(* Logix 5000 project; controller LeakTestAuto vendor 1 type 14 code 226 rev 37.11; software revision 37.01; part 7 of 13 *)
(* tags used below, declared in another part *)
   AOI_CTS1 : AOI_CTS_INSTRUMENT;
   AOI_CTS2 : AOI_CTS_INSTRUMENT;
   AOI_RobotPos : AOI_RobotPositions;
   AOI_SeqSteps : AOI_StandardSeqSteps;
   Conveyor : udt_OutputStructure;
   Conveyor_Seq : udt_SequenceStructure_X64;
   CurrentDUTData : udt_DUTHistory[2];
   DryCycle_N1Ready : BOOL;
   DryCycle_N2Ready : BOOL;
   DUTHistoryDump : udt_DUTHistory;
   DUTTestHistory : udt_DUTHistory[10];
   FFLU_DUTHistory : CONTROL;
   LeakTester1 : udt_OutputStructure;
   LeakTester2 : udt_OutputStructure;
   Nest2Cylinder : udt_OutputStructure;
   OP220 : udt_Mode;
   OP220_Seq : udt_SequenceStructure_X64;
   OutfeedCounter : COUNTER;
   Robot : udt_OutputStructure;
   RobotGripper : udt_OutputStructure;
   RobotInputs : udt_EpsonInputs;
   TON_FailChute : TIMER[10];
   Delay_TMR : TIMER[11];   // Delay Timers
   I_OP220_N3_CONVEYOR_LOAD : ALIAS FOR Local:3:I.Pt12.Data;
   I_OP220_N3_DUT_PRE_NEST_1 : ALIAS FOR Local:3:I.Pt01.Data;
   I_OP220_N3_DUT_PRE_NEST_2 : ALIAS FOR Local:3:I.Pt02.Data;
   I_OP220_N3_NEST2_EXTEND : ALIAS FOR Local:3:I.Pt06.Data;
   I_OP220_N3_REJECT_BIN_OK : ALIAS FOR Local:3:I.Pt09.Data;
   I_OP220_N3_REJECT_CHUTE_PART : ALIAS FOR Local:3:I.Pt10.Data;
   Ignition_Bypass : BOOL;
   James_Dint : DINT;   // James Test Word
   null : STRING;
   ST1_Ignition_DataReady : BOOL;
   ST1_Ignition_DataReady_Setup : BOOL;
   ST1_Ignition_DataReceived : BOOL;
   ST1_Ignition_SerialNum : STRING;
   ST1_Ignition_Status : DINT;
   ST2_Ignition_DataReady : BOOL;
   ST2_Ignition_DataReady_Setup : BOOL;
   ST2_Ignition_DataReceived : BOOL;
   ST2_Ignition_SerialNum : STRING;
   ST2_Ignition_Status : DINT;
(* MainProgram, continued *)

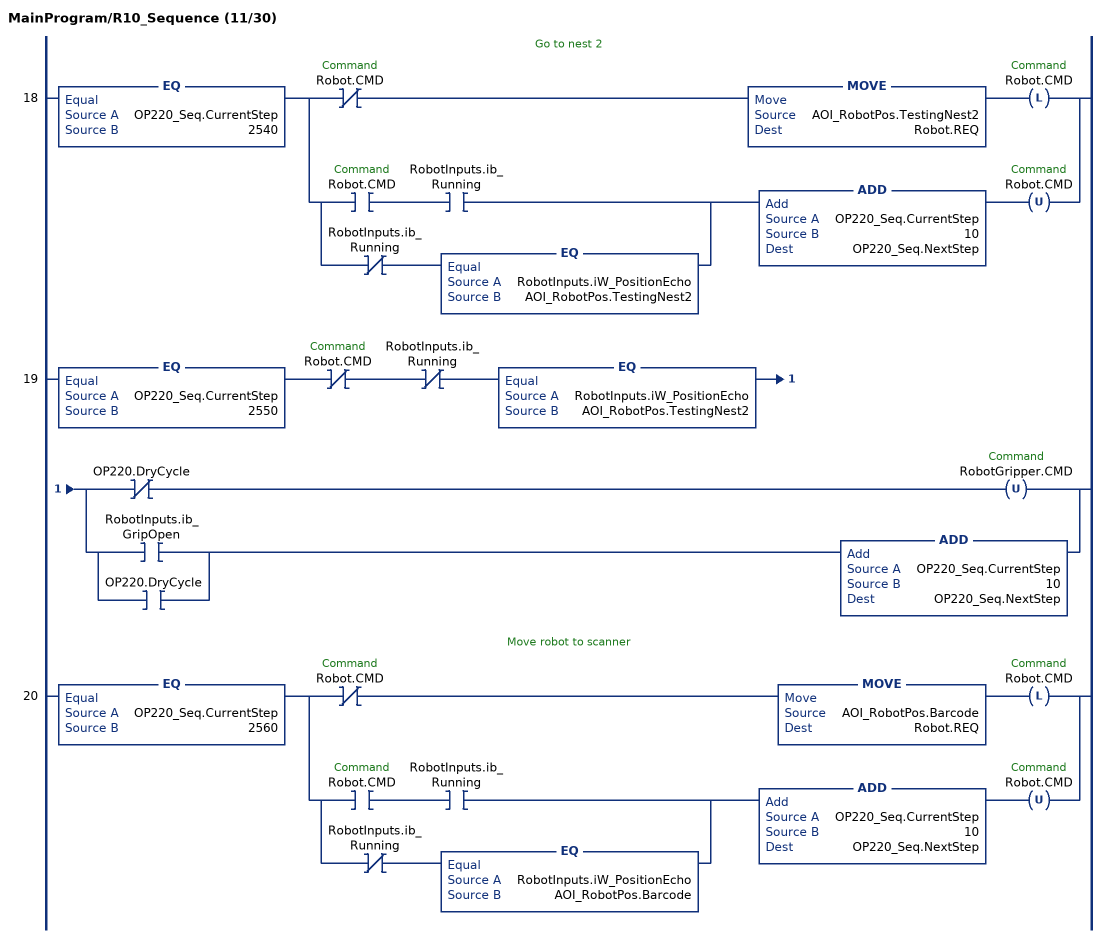
   [picture p74: MainProgram/R10_Sequence rungs 18-20]
   // Go to nest 2
   18: EQ(OP220_Seq.CurrentStep,2540)[XIO(Robot.CMD) MOVE(AOI_RobotPos.TestingNest2,Robot.REQ) OTL(Robot.CMD) ,[XIC(Robot.CMD) XIC(RobotInputs.ib_Running) ,XIO(RobotInputs.ib_Running) EQ(RobotInputs.iW_PositionEcho,AOI_RobotPos.TestingNest2) ] ADD(OP220_Seq.CurrentStep,10,OP220_Seq.NextStep) OTU(Robot.CMD) ];
   19: EQ(OP220_Seq.CurrentStep,2550)XIO(Robot.CMD)XIO(RobotInputs.ib_Running)EQ(RobotInputs.iW_PositionEcho,AOI_RobotPos.TestingNest2)[XIO(OP220.DryCycle) OTU(RobotGripper.CMD) ,[XIC(RobotInputs.ib_GripOpen) ,XIC(OP220.DryCycle) ] ADD(OP220_Seq.CurrentStep,10,OP220_Seq.NextStep) ];
   // Move robot to scanner
   20: EQ(OP220_Seq.CurrentStep,2560)[XIO(Robot.CMD) MOVE(AOI_RobotPos.Barcode,Robot.REQ) OTL(Robot.CMD) ,[XIC(Robot.CMD) XIC(RobotInputs.ib_Running) ,XIO(RobotInputs.ib_Running) EQ(RobotInputs.iW_PositionEcho,AOI_RobotPos.Barcode) ] ADD(OP220_Seq.CurrentStep,10,OP220_Seq.NextStep) OTU(Robot.CMD) ];
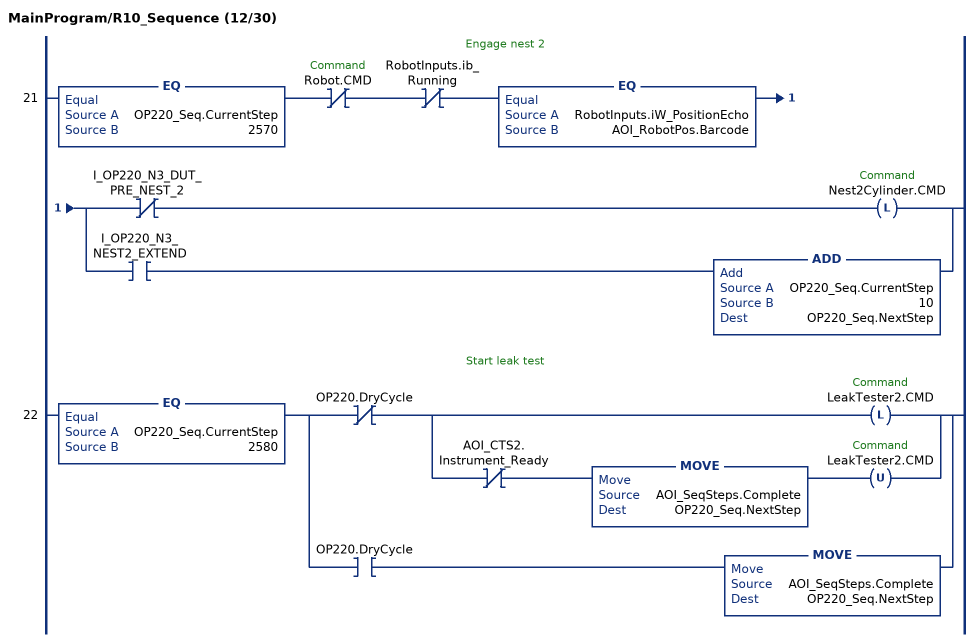
   // Engage nest 2
   21: EQ(OP220_Seq.CurrentStep,2570)XIO(Robot.CMD)XIO(RobotInputs.ib_Running)EQ(RobotInputs.iW_PositionEcho,AOI_RobotPos.Barcode)[XIO(I_OP220_N3_DUT_PRE_NEST_2) OTL(Nest2Cylinder.CMD) ,XIC(I_OP220_N3_NEST2_EXTEND) ADD(OP220_Seq.CurrentStep,10,OP220_Seq.NextStep) ];
   // Start leak test
   22: EQ(OP220_Seq.CurrentStep,2580)[XIO(OP220.DryCycle) [OTL(LeakTester2.CMD) ,XIO(AOI_CTS2.Instrument_Ready) MOVE(AOI_SeqSteps.Complete,OP220_Seq.NextStep) OTU(LeakTester2.CMD) ] ,XIC(OP220.DryCycle) MOVE(AOI_SeqSteps.Complete,OP220_Seq.NextStep) ];
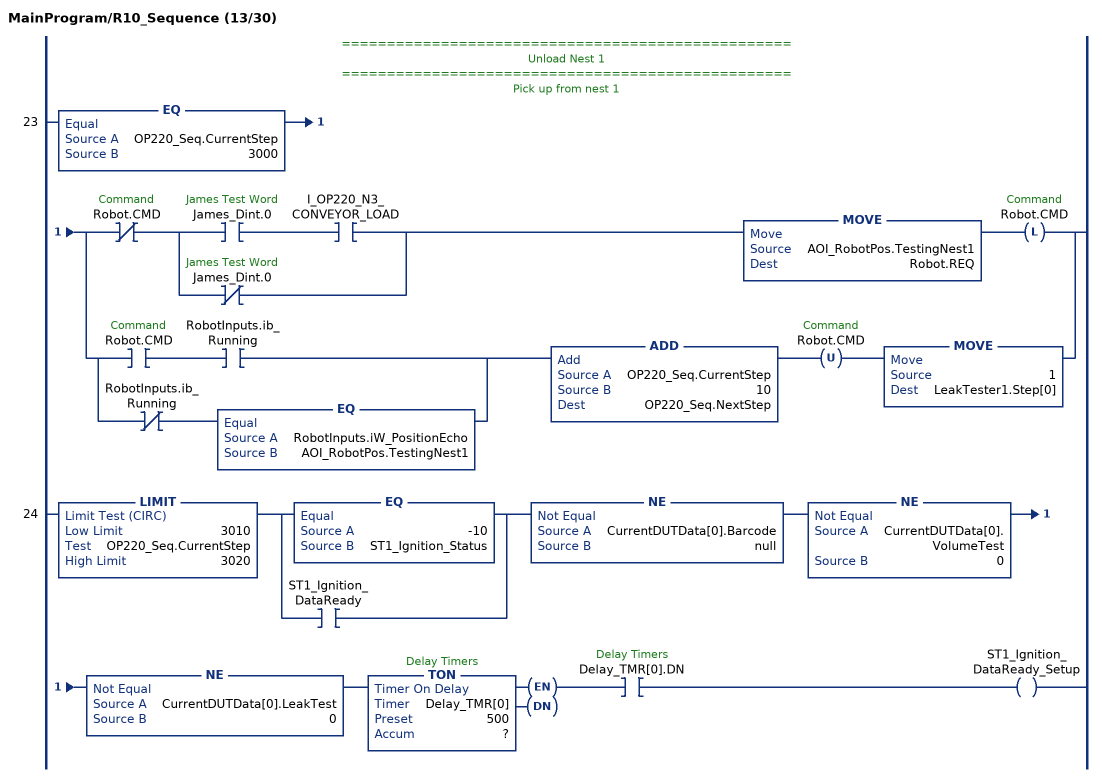
   // ==================================================
   // Unload Nest 1
   // ==================================================
   // Pick up from nest 1
   23: EQ(OP220_Seq.CurrentStep,3000)[XIO(Robot.CMD) [XIC(James_Dint.0) XIC(I_OP220_N3_CONVEYOR_LOAD) ,XIO(James_Dint.0) ] MOVE(AOI_RobotPos.TestingNest1,Robot.REQ) OTL(Robot.CMD) ,[XIC(Robot.CMD) XIC(RobotInputs.ib_Running) ,XIO(RobotInputs.ib_Running) EQ(RobotInputs.iW_PositionEcho,AOI_RobotPos.TestingNest1) ] ADD(OP220_Seq.CurrentStep,10,OP220_Seq.NextStep) OTU(Robot.CMD) MOVE(1,LeakTester1.Step[0]) ];
   24: LIMIT(3010,OP220_Seq.CurrentStep,3020)[EQ(-10,ST1_Ignition_Status) ,XIC(ST1_Ignition_DataReady) ]NE(CurrentDUTData[0].Barcode,null)NE(CurrentDUTData[0].VolumeTest,0)NE(CurrentDUTData[0].LeakTest,0)TON(Delay_TMR[0],?,?)XIC(Delay_TMR[0].DN)OTE(ST1_Ignition_DataReady_Setup);
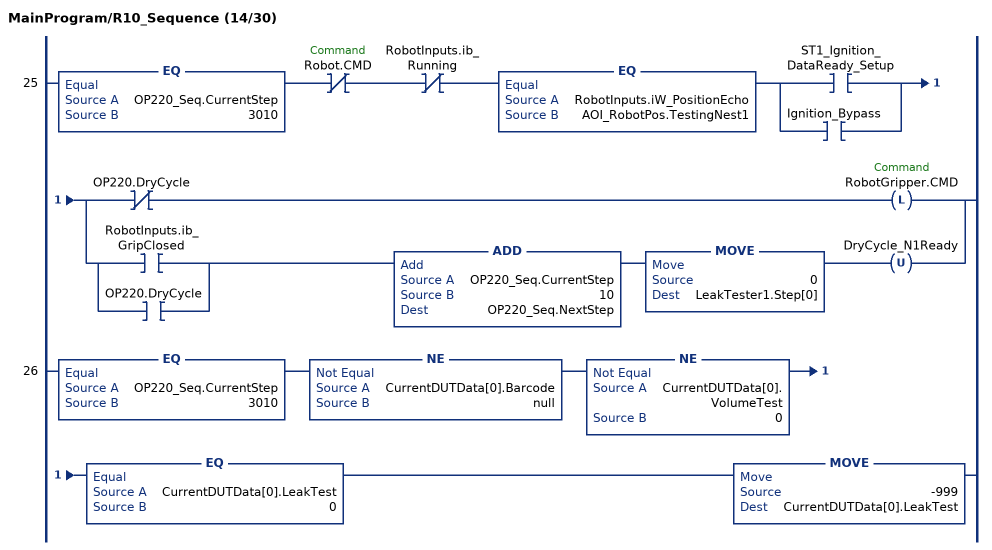
   25: EQ(OP220_Seq.CurrentStep,3010)XIO(Robot.CMD)XIO(RobotInputs.ib_Running)EQ(RobotInputs.iW_PositionEcho,AOI_RobotPos.TestingNest1)[XIC(ST1_Ignition_DataReady_Setup) ,XIC(Ignition_Bypass) ][XIO(OP220.DryCycle) OTL(RobotGripper.CMD) ,[XIC(RobotInputs.ib_GripClosed) ,XIC(OP220.DryCycle) ] ADD(OP220_Seq.CurrentStep,10,OP220_Seq.NextStep) MOVE(0,LeakTester1.Step[0]) OTU(DryCycle_N1Ready) ];
   26: EQ(OP220_Seq.CurrentStep,3010)NE(CurrentDUTData[0].Barcode,null)NE(CurrentDUTData[0].VolumeTest,0)EQ(CurrentDUTData[0].LeakTest,0)MOVE(-999,CurrentDUTData[0].LeakTest);
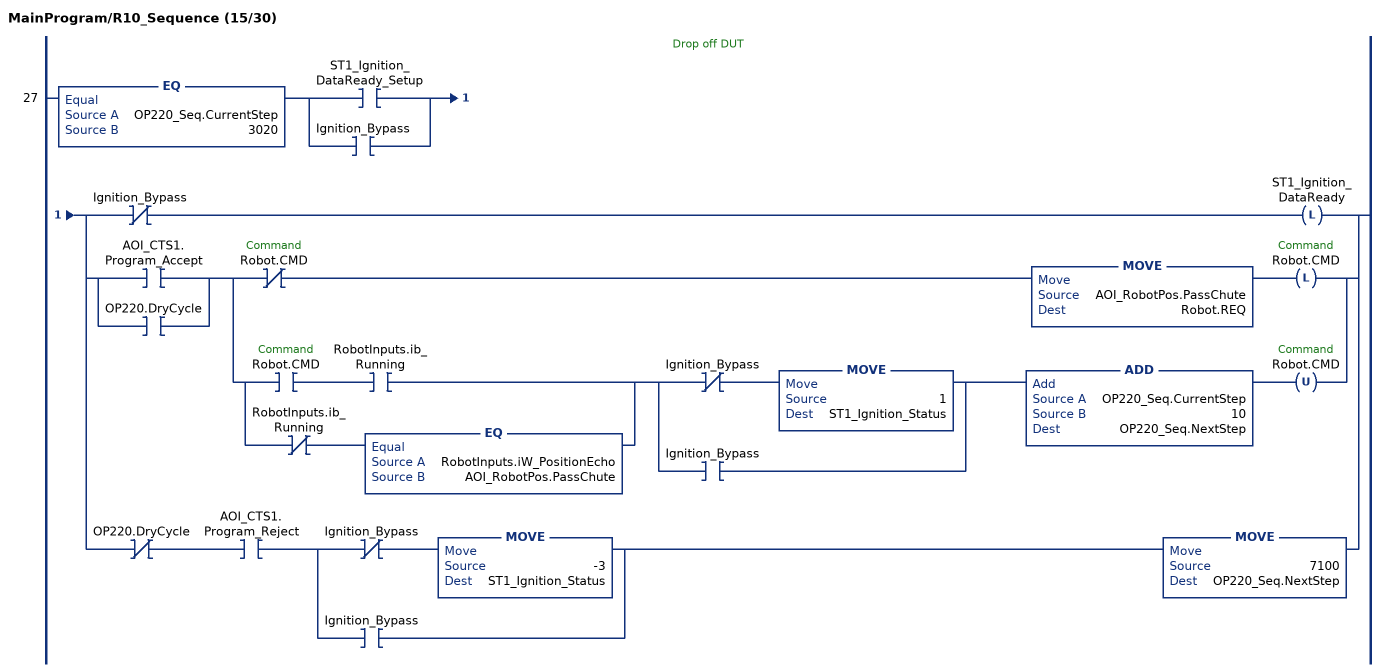
   // Drop off DUT
   27: EQ(OP220_Seq.CurrentStep,3020)[XIC(ST1_Ignition_DataReady_Setup) ,XIC(Ignition_Bypass) ][XIO(Ignition_Bypass) OTL(ST1_Ignition_DataReady) ,[XIC(AOI_CTS1.Program_Accept) ,XIC(OP220.DryCycle) ] [XIO(Robot.CMD) MOVE(AOI_RobotPos.PassChute,Robot.REQ) OTL(Robot.CMD) ,[XIC(Robot.CMD) XIC(RobotInputs.ib_Running) ,XIO(RobotInputs.ib_Running) EQ(RobotInputs.iW_PositionEcho,AOI_RobotPos.PassChute) ] [XIO(Ignition_Bypass) MOVE(1,ST1_Ignition_Status) ,XIC(Ignition_Bypass) ] ADD(OP220_Seq.CurrentStep,10,OP220_Seq.NextStep) OTU(Robot.CMD) ] ,XIO(OP220.DryCycle) XIC(AOI_CTS1.Program_Reject) [XIO(Ignition_Bypass) MOVE(-3,ST1_Ignition_Status) ,XIC(Ignition_Bypass) ] MOVE(7100,OP220_Seq.NextStep) ];
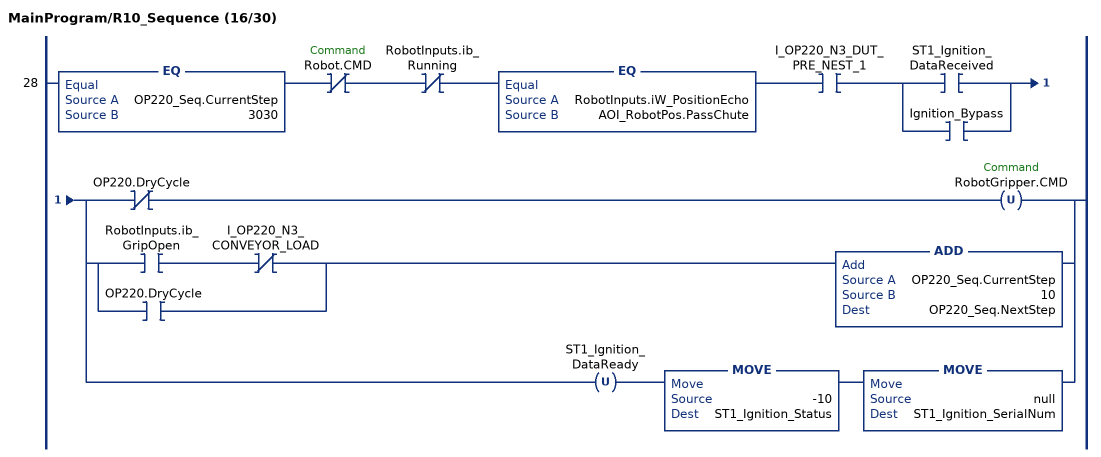
   28: EQ(OP220_Seq.CurrentStep,3030)XIO(Robot.CMD)XIO(RobotInputs.ib_Running)EQ(RobotInputs.iW_PositionEcho,AOI_RobotPos.PassChute)XIC(I_OP220_N3_DUT_PRE_NEST_1)[XIC(ST1_Ignition_DataReceived) ,XIC(Ignition_Bypass) ][XIO(OP220.DryCycle) OTU(RobotGripper.CMD) ,[XIC(RobotInputs.ib_GripOpen) XIO(I_OP220_N3_CONVEYOR_LOAD) ,XIC(OP220.DryCycle) ] ADD(OP220_Seq.CurrentStep,10,OP220_Seq.NextStep) ,OTU(ST1_Ignition_DataReady) MOVE(-10,ST1_Ignition_Status) MOVE(null,ST1_Ignition_SerialNum) ];
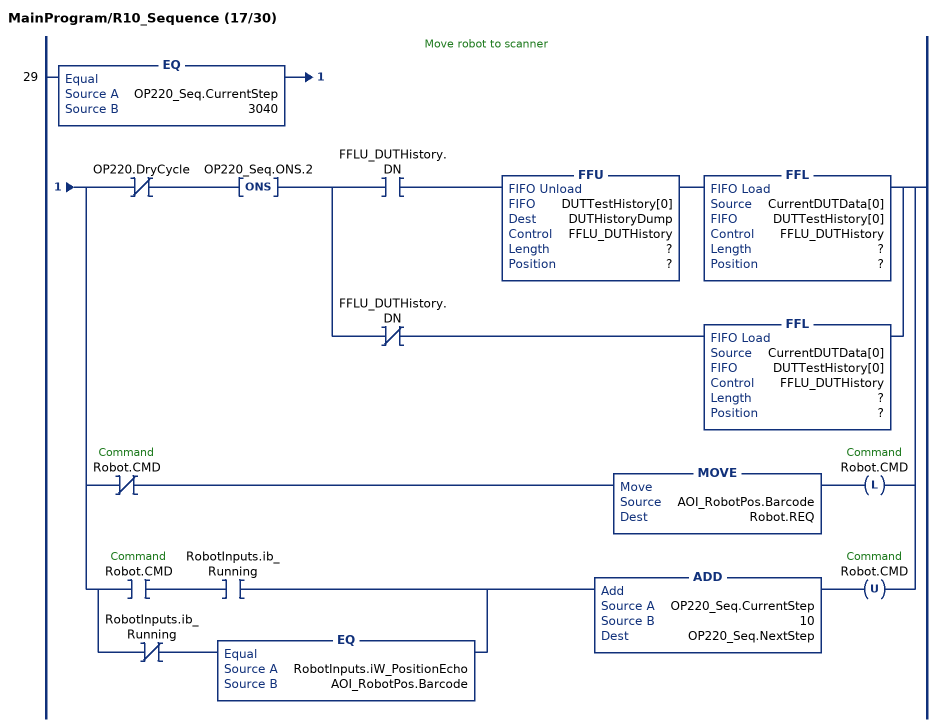
   // Move robot to scanner
   29: EQ(OP220_Seq.CurrentStep,3040)[XIO(OP220.DryCycle) ONS(OP220_Seq.ONS.2) [XIC(FFLU_DUTHistory.DN) FFU(DUTTestHistory[0],DUTHistoryDump,FFLU_DUTHistory,?,?) FFL(CurrentDUTData[0],DUTTestHistory[0],FFLU_DUTHistory,?,?) ,XIO(FFLU_DUTHistory.DN) FFL(CurrentDUTData[0],DUTTestHistory[0],FFLU_DUTHistory,?,?) ] ,XIO(Robot.CMD) MOVE(AOI_RobotPos.Barcode,Robot.REQ) OTL(Robot.CMD) ,[XIC(Robot.CMD) XIC(RobotInputs.ib_Running) ,XIO(RobotInputs.ib_Running) EQ(RobotInputs.iW_PositionEcho,AOI_RobotPos.Barcode) ] ADD(OP220_Seq.CurrentStep,10,OP220_Seq.NextStep) OTU(Robot.CMD) ];
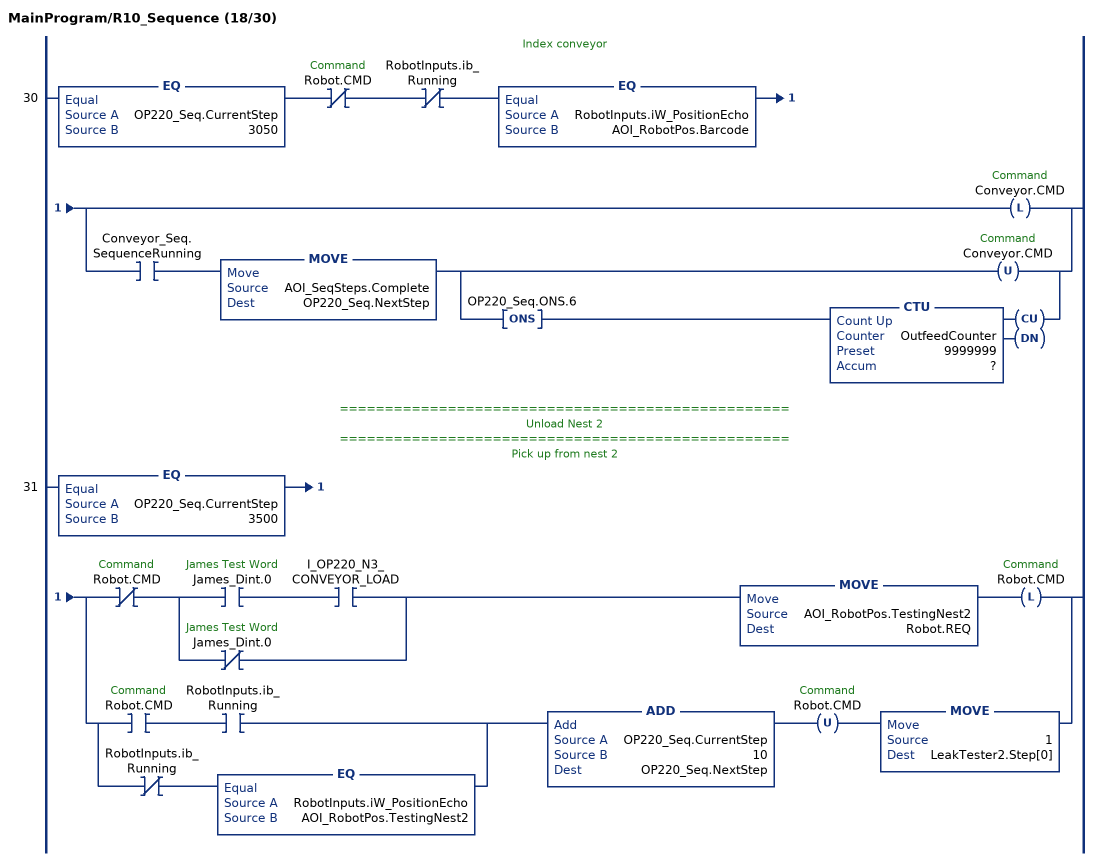
   // Index conveyor
   30: EQ(OP220_Seq.CurrentStep,3050)XIO(Robot.CMD)XIO(RobotInputs.ib_Running)EQ(RobotInputs.iW_PositionEcho,AOI_RobotPos.Barcode)[OTL(Conveyor.CMD) ,XIC(Conveyor_Seq.SequenceRunning) MOVE(AOI_SeqSteps.Complete,OP220_Seq.NextStep) [OTU(Conveyor.CMD) ,ONS(OP220_Seq.ONS.6) CTU(OutfeedCounter,?,?) ] ];
   // ==================================================
   // Unload Nest 2
   // ==================================================
   // Pick up from nest 2
   31: EQ(OP220_Seq.CurrentStep,3500)[XIO(Robot.CMD) [XIC(James_Dint.0) XIC(I_OP220_N3_CONVEYOR_LOAD) ,XIO(James_Dint.0) ] MOVE(AOI_RobotPos.TestingNest2,Robot.REQ) OTL(Robot.CMD) ,[XIC(Robot.CMD) XIC(RobotInputs.ib_Running) ,XIO(RobotInputs.ib_Running) EQ(RobotInputs.iW_PositionEcho,AOI_RobotPos.TestingNest2) ] ADD(OP220_Seq.CurrentStep,10,OP220_Seq.NextStep) OTU(Robot.CMD) MOVE(1,LeakTester2.Step[0]) ];
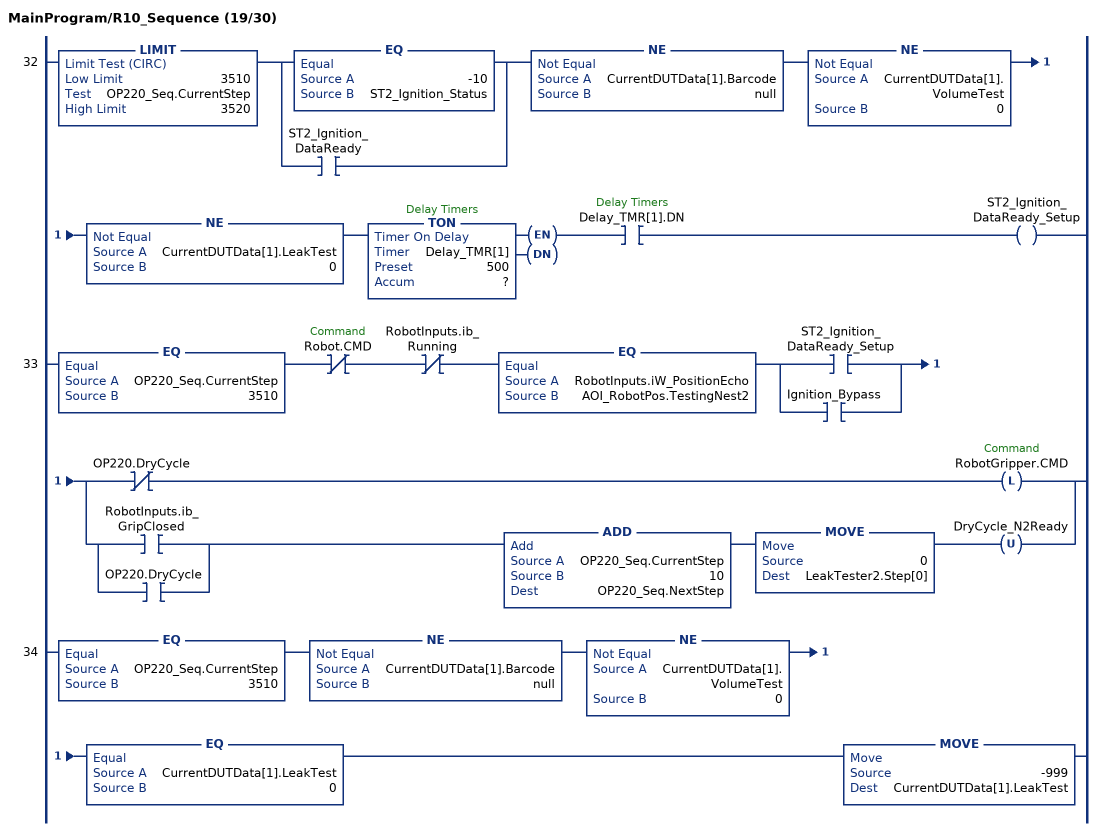
   32: LIMIT(3510,OP220_Seq.CurrentStep,3520)[EQ(-10,ST2_Ignition_Status) ,XIC(ST2_Ignition_DataReady) ]NE(CurrentDUTData[1].Barcode,null)NE(CurrentDUTData[1].VolumeTest,0)NE(CurrentDUTData[1].LeakTest,0)TON(Delay_TMR[1],?,?)XIC(Delay_TMR[1].DN)OTE(ST2_Ignition_DataReady_Setup);
   33: EQ(OP220_Seq.CurrentStep,3510)XIO(Robot.CMD)XIO(RobotInputs.ib_Running)EQ(RobotInputs.iW_PositionEcho,AOI_RobotPos.TestingNest2)[XIC(ST2_Ignition_DataReady_Setup) ,XIC(Ignition_Bypass) ][XIO(OP220.DryCycle) OTL(RobotGripper.CMD) ,[XIC(RobotInputs.ib_GripClosed) ,XIC(OP220.DryCycle) ] ADD(OP220_Seq.CurrentStep,10,OP220_Seq.NextStep) MOVE(0,LeakTester2.Step[0]) OTU(DryCycle_N2Ready) ];
   34: EQ(OP220_Seq.CurrentStep,3510)NE(CurrentDUTData[1].Barcode,null)NE(CurrentDUTData[1].VolumeTest,0)EQ(CurrentDUTData[1].LeakTest,0)MOVE(-999,CurrentDUTData[1].LeakTest);
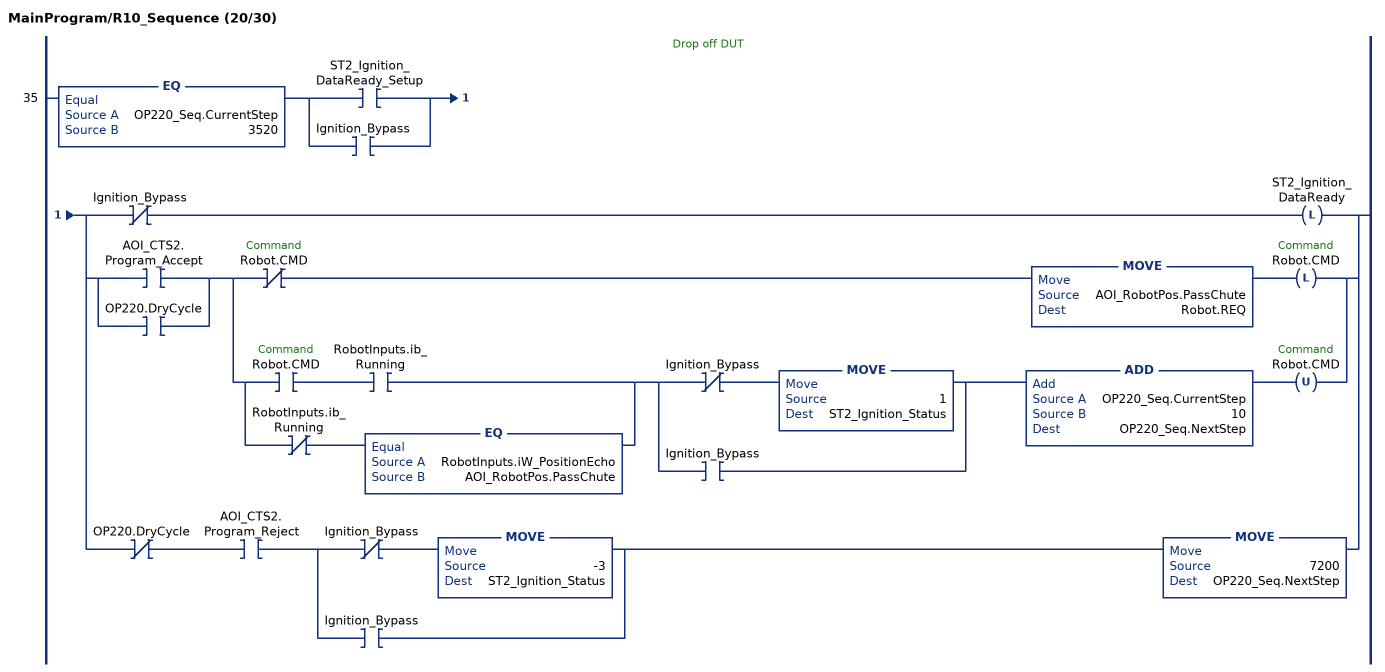
   // Drop off DUT
   35: EQ(OP220_Seq.CurrentStep,3520)[XIC(ST2_Ignition_DataReady_Setup) ,XIC(Ignition_Bypass) ][XIO(Ignition_Bypass) OTL(ST2_Ignition_DataReady) ,[XIC(AOI_CTS2.Program_Accept) ,XIC(OP220.DryCycle) ] [XIO(Robot.CMD) MOVE(AOI_RobotPos.PassChute,Robot.REQ) OTL(Robot.CMD) ,[XIC(Robot.CMD) XIC(RobotInputs.ib_Running) ,XIO(RobotInputs.ib_Running) EQ(RobotInputs.iW_PositionEcho,AOI_RobotPos.PassChute) ] [XIO(Ignition_Bypass) MOVE(1,ST2_Ignition_Status) ,XIC(Ignition_Bypass) ] ADD(OP220_Seq.CurrentStep,10,OP220_Seq.NextStep) OTU(Robot.CMD) ] ,XIO(OP220.DryCycle) XIC(AOI_CTS2.Program_Reject) [XIO(Ignition_Bypass) MOVE(-3,ST2_Ignition_Status) ,XIC(Ignition_Bypass) ] MOVE(7200,OP220_Seq.NextStep) ];
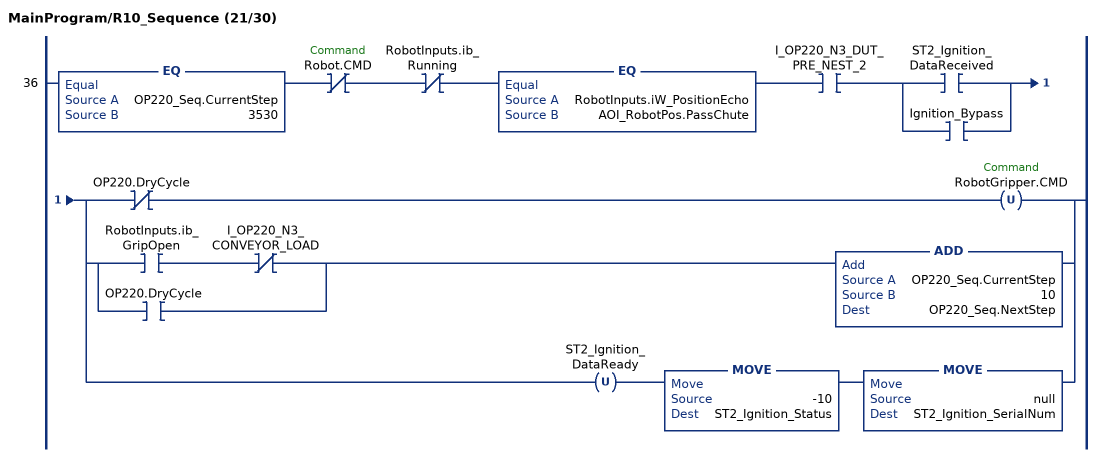
   36: EQ(OP220_Seq.CurrentStep,3530)XIO(Robot.CMD)XIO(RobotInputs.ib_Running)EQ(RobotInputs.iW_PositionEcho,AOI_RobotPos.PassChute)XIC(I_OP220_N3_DUT_PRE_NEST_2)[XIC(ST2_Ignition_DataReceived) ,XIC(Ignition_Bypass) ][XIO(OP220.DryCycle) OTU(RobotGripper.CMD) ,[XIC(RobotInputs.ib_GripOpen) XIO(I_OP220_N3_CONVEYOR_LOAD) ,XIC(OP220.DryCycle) ] ADD(OP220_Seq.CurrentStep,10,OP220_Seq.NextStep) ,OTU(ST2_Ignition_DataReady) MOVE(-10,ST2_Ignition_Status) MOVE(null,ST2_Ignition_SerialNum) ];
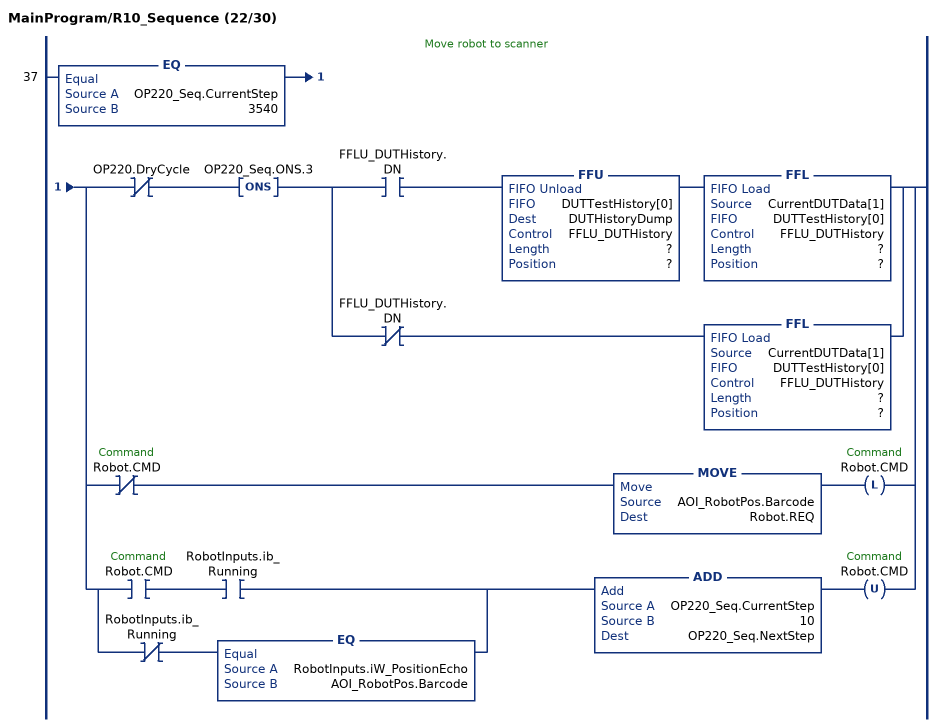
   // Move robot to scanner
   37: EQ(OP220_Seq.CurrentStep,3540)[XIO(OP220.DryCycle) ONS(OP220_Seq.ONS.3) [XIC(FFLU_DUTHistory.DN) FFU(DUTTestHistory[0],DUTHistoryDump,FFLU_DUTHistory,?,?) FFL(CurrentDUTData[1],DUTTestHistory[0],FFLU_DUTHistory,?,?) ,XIO(FFLU_DUTHistory.DN) FFL(CurrentDUTData[1],DUTTestHistory[0],FFLU_DUTHistory,?,?) ] ,XIO(Robot.CMD) MOVE(AOI_RobotPos.Barcode,Robot.REQ) OTL(Robot.CMD) ,[XIC(Robot.CMD) XIC(RobotInputs.ib_Running) ,XIO(RobotInputs.ib_Running) EQ(RobotInputs.iW_PositionEcho,AOI_RobotPos.Barcode) ] ADD(OP220_Seq.CurrentStep,10,OP220_Seq.NextStep) OTU(Robot.CMD) ];
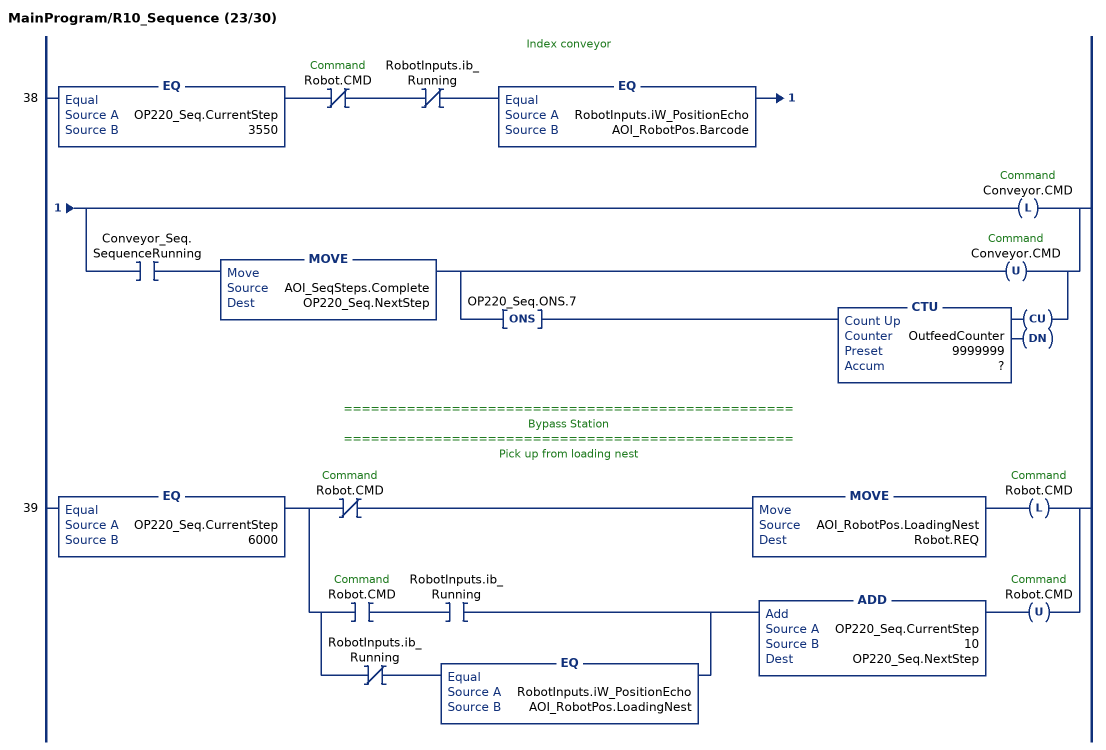
   // Index conveyor
   38: EQ(OP220_Seq.CurrentStep,3550)XIO(Robot.CMD)XIO(RobotInputs.ib_Running)EQ(RobotInputs.iW_PositionEcho,AOI_RobotPos.Barcode)[OTL(Conveyor.CMD) ,XIC(Conveyor_Seq.SequenceRunning) MOVE(AOI_SeqSteps.Complete,OP220_Seq.NextStep) [OTU(Conveyor.CMD) ,ONS(OP220_Seq.ONS.7) CTU(OutfeedCounter,?,?) ] ];
   // ==================================================
   // Bypass Station
   // ==================================================
   // Pick up from loading nest
   39: EQ(OP220_Seq.CurrentStep,6000)[XIO(Robot.CMD) MOVE(AOI_RobotPos.LoadingNest,Robot.REQ) OTL(Robot.CMD) ,[XIC(Robot.CMD) XIC(RobotInputs.ib_Running) ,XIO(RobotInputs.ib_Running) EQ(RobotInputs.iW_PositionEcho,AOI_RobotPos.LoadingNest) ] ADD(OP220_Seq.CurrentStep,10,OP220_Seq.NextStep) OTU(Robot.CMD) ];
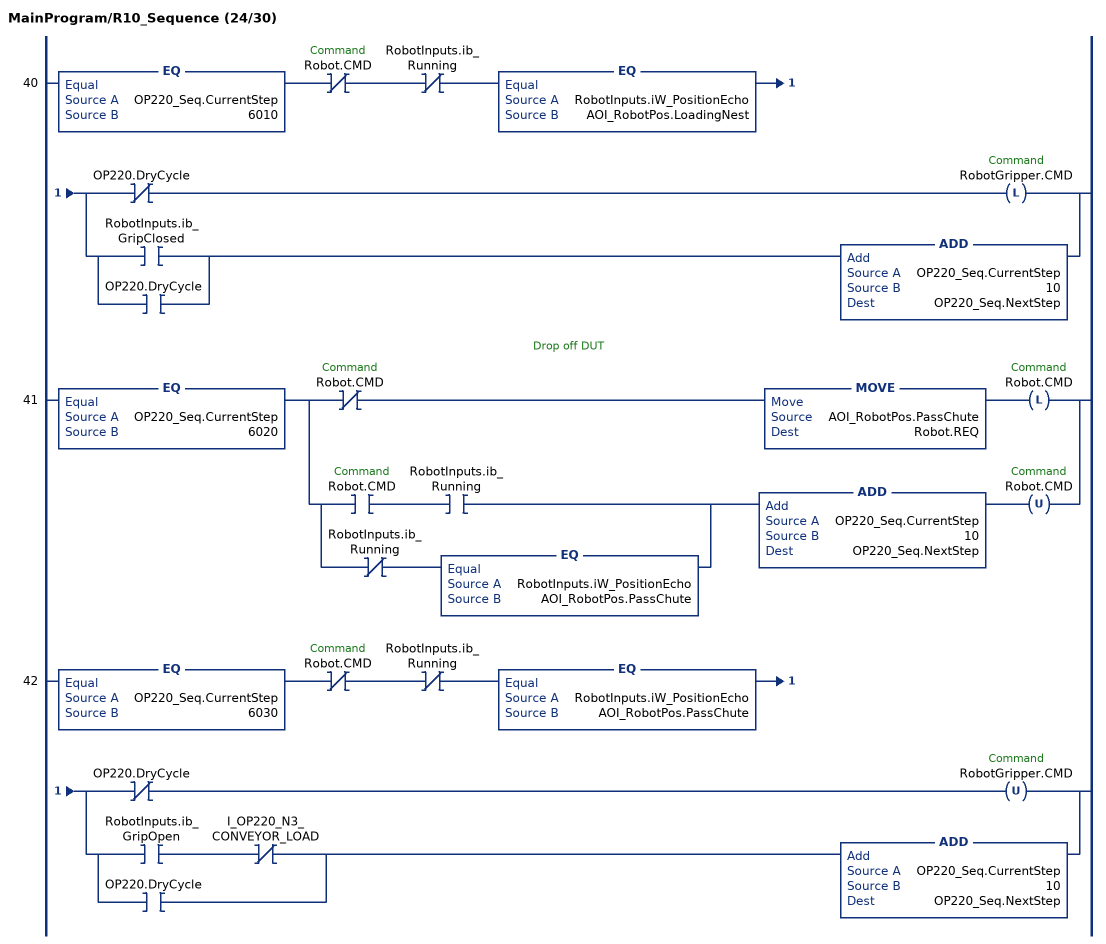
   40: EQ(OP220_Seq.CurrentStep,6010)XIO(Robot.CMD)XIO(RobotInputs.ib_Running)EQ(RobotInputs.iW_PositionEcho,AOI_RobotPos.LoadingNest)[XIO(OP220.DryCycle) OTL(RobotGripper.CMD) ,[XIC(RobotInputs.ib_GripClosed) ,XIC(OP220.DryCycle) ] ADD(OP220_Seq.CurrentStep,10,OP220_Seq.NextStep) ];
   // Drop off DUT
   41: EQ(OP220_Seq.CurrentStep,6020)[XIO(Robot.CMD) MOVE(AOI_RobotPos.PassChute,Robot.REQ) OTL(Robot.CMD) ,[XIC(Robot.CMD) XIC(RobotInputs.ib_Running) ,XIO(RobotInputs.ib_Running) EQ(RobotInputs.iW_PositionEcho,AOI_RobotPos.PassChute) ] ADD(OP220_Seq.CurrentStep,10,OP220_Seq.NextStep) OTU(Robot.CMD) ];
   42: EQ(OP220_Seq.CurrentStep,6030)XIO(Robot.CMD)XIO(RobotInputs.ib_Running)EQ(RobotInputs.iW_PositionEcho,AOI_RobotPos.PassChute)[XIO(OP220.DryCycle) OTU(RobotGripper.CMD) ,[XIC(RobotInputs.ib_GripOpen) XIO(I_OP220_N3_CONVEYOR_LOAD) ,XIC(OP220.DryCycle) ] ADD(OP220_Seq.CurrentStep,10,OP220_Seq.NextStep) ];
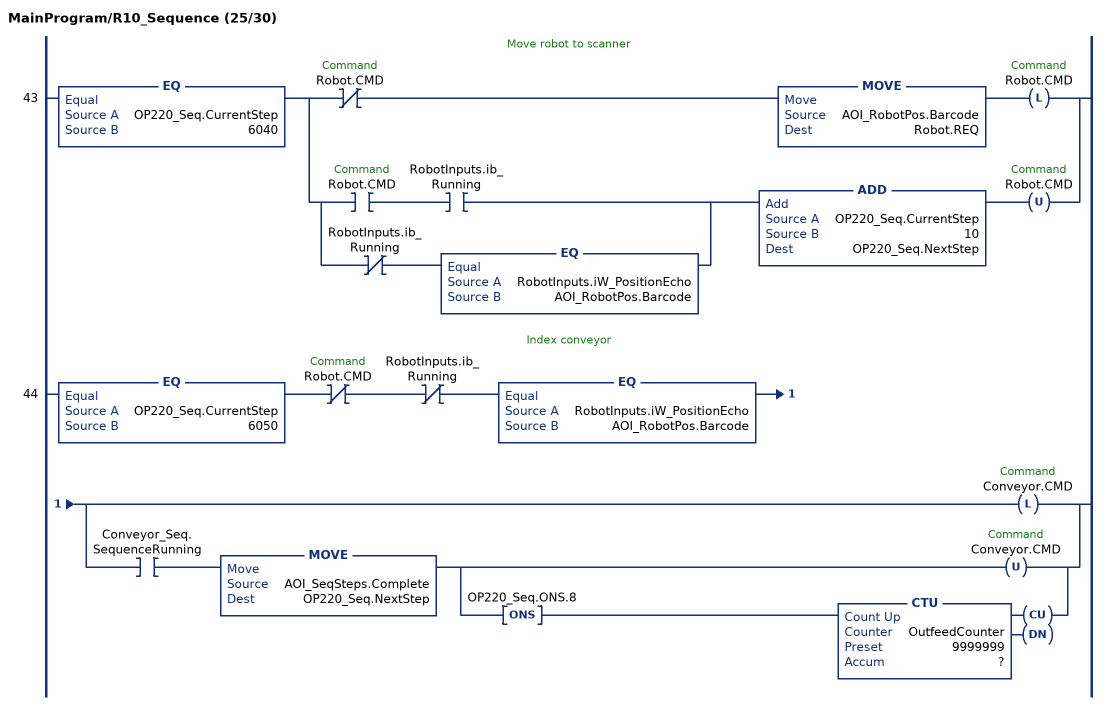
   // Move robot to scanner
   43: EQ(OP220_Seq.CurrentStep,6040)[XIO(Robot.CMD) MOVE(AOI_RobotPos.Barcode,Robot.REQ) OTL(Robot.CMD) ,[XIC(Robot.CMD) XIC(RobotInputs.ib_Running) ,XIO(RobotInputs.ib_Running) EQ(RobotInputs.iW_PositionEcho,AOI_RobotPos.Barcode) ] ADD(OP220_Seq.CurrentStep,10,OP220_Seq.NextStep) OTU(Robot.CMD) ];
   // Index conveyor
   44: EQ(OP220_Seq.CurrentStep,6050)XIO(Robot.CMD)XIO(RobotInputs.ib_Running)EQ(RobotInputs.iW_PositionEcho,AOI_RobotPos.Barcode)[OTL(Conveyor.CMD) ,XIC(Conveyor_Seq.SequenceRunning) MOVE(AOI_SeqSteps.Complete,OP220_Seq.NextStep) [OTU(Conveyor.CMD) ,ONS(OP220_Seq.ONS.8) CTU(OutfeedCounter,?,?) ] ];
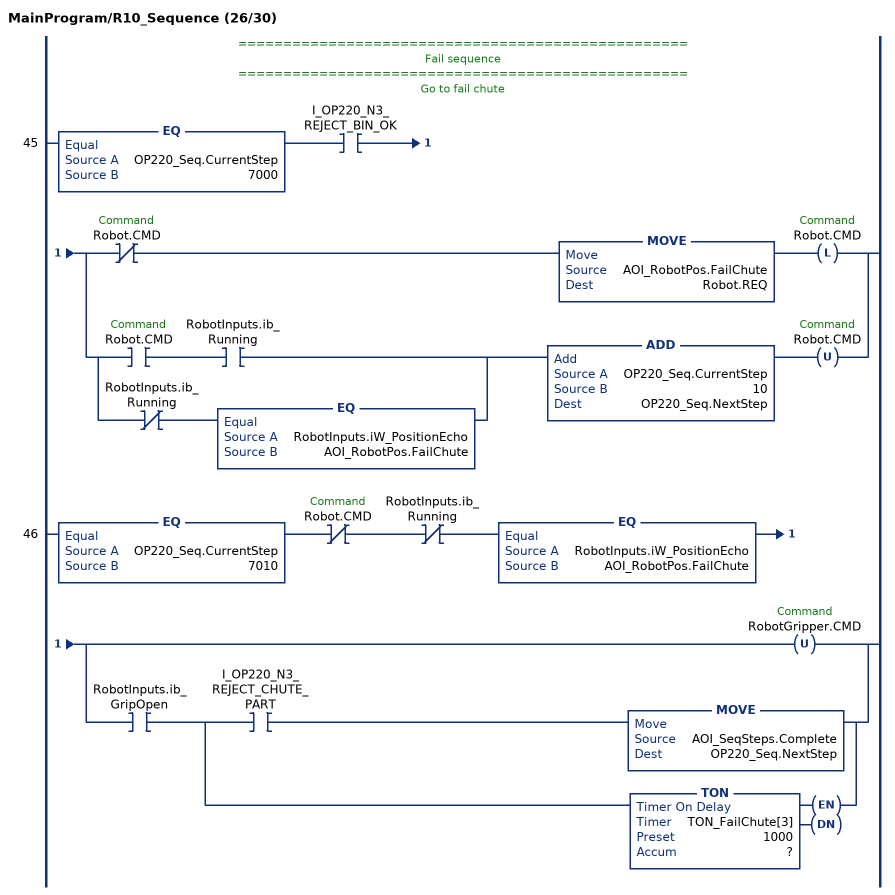
   // ==================================================
   // Fail sequence
   // ==================================================
   // Go to fail chute
   45: EQ(OP220_Seq.CurrentStep,7000)XIC(I_OP220_N3_REJECT_BIN_OK)[XIO(Robot.CMD) MOVE(AOI_RobotPos.FailChute,Robot.REQ) OTL(Robot.CMD) ,[XIC(Robot.CMD) XIC(RobotInputs.ib_Running) ,XIO(RobotInputs.ib_Running) EQ(RobotInputs.iW_PositionEcho,AOI_RobotPos.FailChute) ] ADD(OP220_Seq.CurrentStep,10,OP220_Seq.NextStep) OTU(Robot.CMD) ];
   46: EQ(OP220_Seq.CurrentStep,7010)XIO(Robot.CMD)XIO(RobotInputs.ib_Running)EQ(RobotInputs.iW_PositionEcho,AOI_RobotPos.FailChute)[OTU(RobotGripper.CMD) ,XIC(RobotInputs.ib_GripOpen) [XIC(I_OP220_N3_REJECT_CHUTE_PART) MOVE(AOI_SeqSteps.Complete,OP220_Seq.NextStep) ,TON(TON_FailChute[3],?,?) ] ];
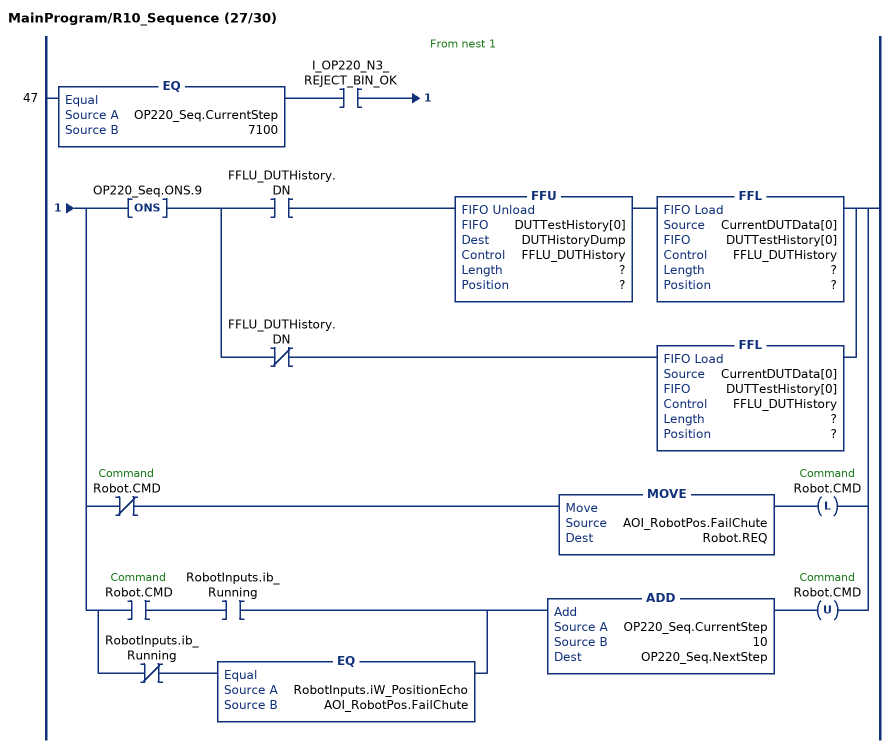
   // From nest 1
   47: EQ(OP220_Seq.CurrentStep,7100)XIC(I_OP220_N3_REJECT_BIN_OK)[ONS(OP220_Seq.ONS.9) [XIC(FFLU_DUTHistory.DN) FFU(DUTTestHistory[0],DUTHistoryDump,FFLU_DUTHistory,?,?) FFL(CurrentDUTData[0],DUTTestHistory[0],FFLU_DUTHistory,?,?) ,XIO(FFLU_DUTHistory.DN) FFL(CurrentDUTData[0],DUTTestHistory[0],FFLU_DUTHistory,?,?) ] ,XIO(Robot.CMD) MOVE(AOI_RobotPos.FailChute,Robot.REQ) OTL(Robot.CMD) ,[XIC(Robot.CMD) XIC(RobotInputs.ib_Running) ,XIO(RobotInputs.ib_Running) EQ(RobotInputs.iW_PositionEcho,AOI_RobotPos.FailChute) ] ADD(OP220_Seq.CurrentStep,10,OP220_Seq.NextStep) OTU(Robot.CMD) ];
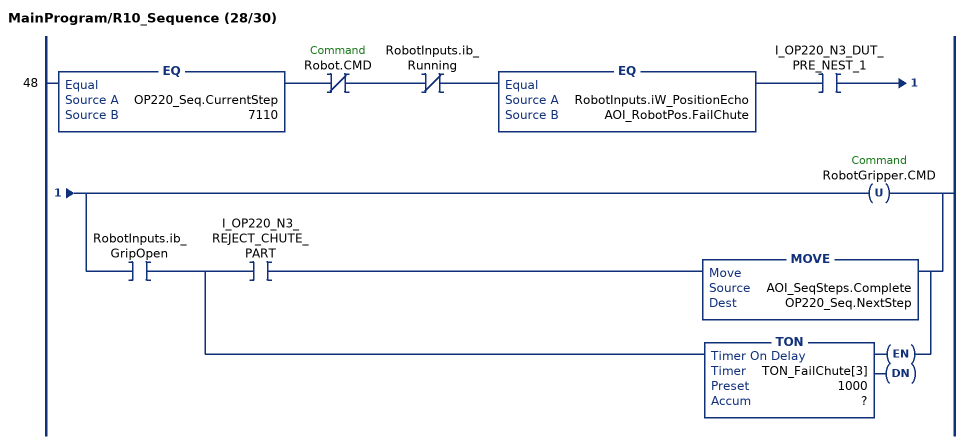
   48: EQ(OP220_Seq.CurrentStep,7110)XIO(Robot.CMD)XIO(RobotInputs.ib_Running)EQ(RobotInputs.iW_PositionEcho,AOI_RobotPos.FailChute)XIC(I_OP220_N3_DUT_PRE_NEST_1)[OTU(RobotGripper.CMD) ,XIC(RobotInputs.ib_GripOpen) [XIC(I_OP220_N3_REJECT_CHUTE_PART) MOVE(AOI_SeqSteps.Complete,OP220_Seq.NextStep) ,TON(TON_FailChute[3],?,?) ] ];
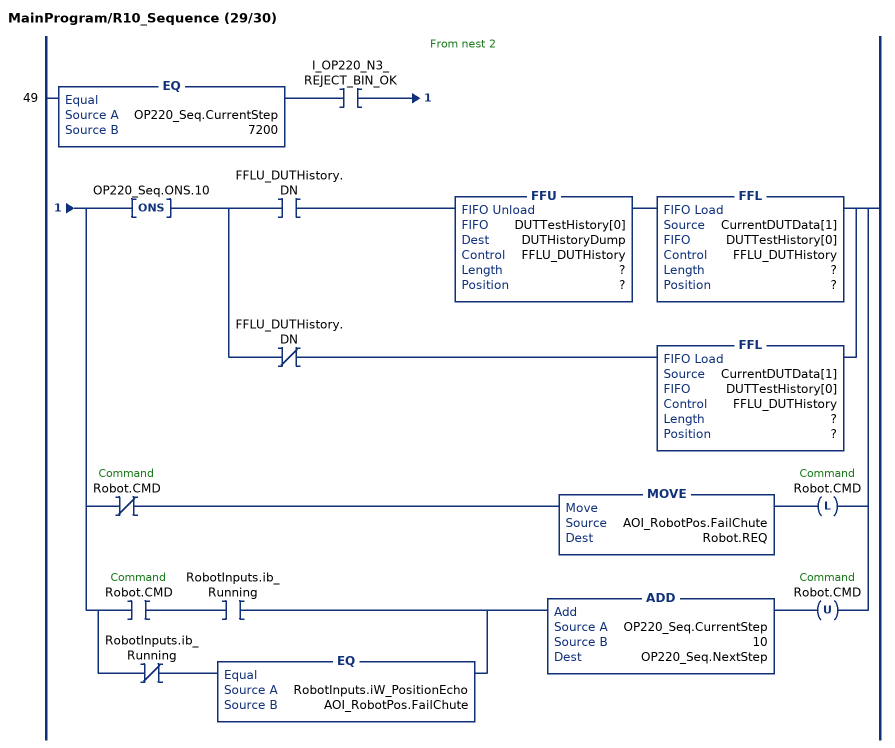
   // From nest 2
   49: EQ(OP220_Seq.CurrentStep,7200)XIC(I_OP220_N3_REJECT_BIN_OK)[ONS(OP220_Seq.ONS.10) [XIC(FFLU_DUTHistory.DN) FFU(DUTTestHistory[0],DUTHistoryDump,FFLU_DUTHistory,?,?) FFL(CurrentDUTData[1],DUTTestHistory[0],FFLU_DUTHistory,?,?) ,XIO(FFLU_DUTHistory.DN) FFL(CurrentDUTData[1],DUTTestHistory[0],FFLU_DUTHistory,?,?) ] ,XIO(Robot.CMD) MOVE(AOI_RobotPos.FailChute,Robot.REQ) OTL(Robot.CMD) ,[XIC(Robot.CMD) XIC(RobotInputs.ib_Running) ,XIO(RobotInputs.ib_Running) EQ(RobotInputs.iW_PositionEcho,AOI_RobotPos.FailChute) ] ADD(OP220_Seq.CurrentStep,10,OP220_Seq.NextStep) OTU(Robot.CMD) ];
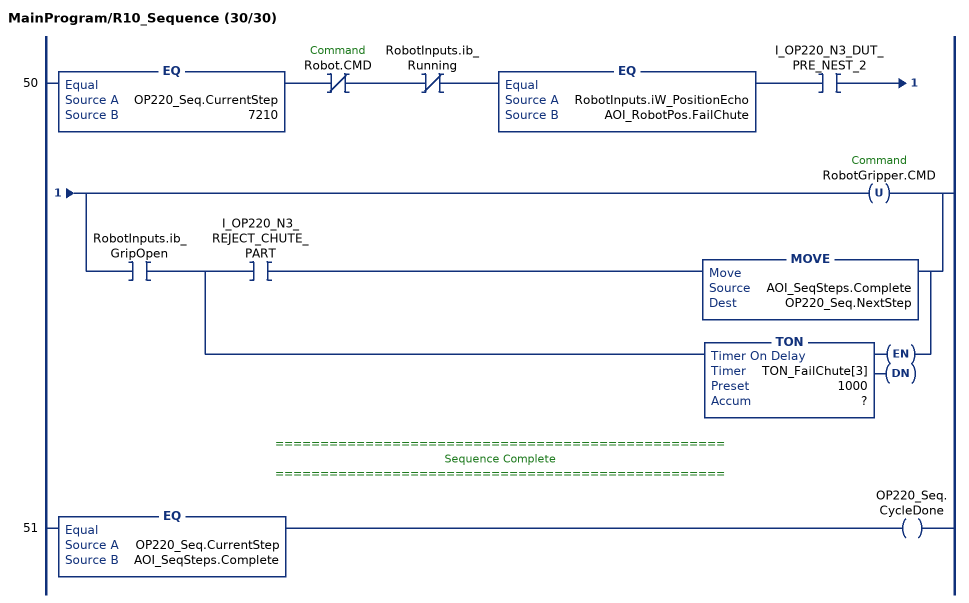
   50: EQ(OP220_Seq.CurrentStep,7210)XIO(Robot.CMD)XIO(RobotInputs.ib_Running)EQ(RobotInputs.iW_PositionEcho,AOI_RobotPos.FailChute)XIC(I_OP220_N3_DUT_PRE_NEST_2)[OTU(RobotGripper.CMD) ,XIC(RobotInputs.ib_GripOpen) [XIC(I_OP220_N3_REJECT_CHUTE_PART) MOVE(AOI_SeqSteps.Complete,OP220_Seq.NextStep) ,TON(TON_FailChute[3],?,?) ] ];
   // ==================================================
   // Sequence Complete
   // ==================================================
   51: EQ(OP220_Seq.CurrentStep,AOI_SeqSteps.Complete)OTE(OP220_Seq.CycleDone);
END_ROUTINE
